PROGRAM EntitiesExample
VAR
END_VAR

ToggleExample();

END_PROGRAM

(* stored: Version 1.1.0.1
   POU EntitiesExample: Id {4b3be423-e5e7-40f1-8b7e-3a07d398763c}, SpecialFunc None *)
